Staubli VAL3: Log.pgx

program Log()
begin
  do
    // Registrar un nou event al logger
    if bNewLog==true
      // Desplaçar registre d'events
      for nLog=49 to 1 step -1
        sLog[nLog]=sLog[nLog-1]
      endFor
      // Afegir nou event
      sLog[0]=sNewLog
      bNewLog=false
    endIf

  until false
end
